// TwinCAT 3 PLC project AD_DA
// ProgramVersion: 3.1.4020.2
// libraries:
//   Tc2_Standard, * (Beckhoff Automation GmbH)
//   Tc2_System, * (Beckhoff Automation GmbH)
//   Tc3_Module, * (Beckhoff Automation GmbH)
// project tree:
//   FB_Lib/FB_ActionneurSimple/ FB_ActionneurSimple.TcPOU, ST_Erreur.TcDUT, ST_ParamActionneur.TcDUT
//   FB_Lib/ FB_analo_and_digital.TcPOU, FB_Etape.TcPOU
//   FB_Lib/FB_GestionModes/ FB_Btn.TcPOU, FB_CycleAuto.TcPOU, FB_CycleInit.TcPOU, FB_CycleMan.TcPOU, FB_MMA.TcPOU, p_InitVar.TcPOU
//   FB_Lib/FB_GestionModes/IO/ ST_IO.TcDUT, ST_IOInput.TcDUT, ST_IOInputSimul.TcDUT, ST_IOOutput.TcDUT, ST_IOOutputSimul.TcDUT
//   FB_Lib/FB_GestionModes/Param/ E_ModeMMA.TcDUT, ST_Param.TcDUT, ST_ParamFixed.TcDUT, ST_ParamRecipe.TcDUT, ST_ParamStatus.TcDUT
//   GVLs/ GVL.TcGVL
//   / PlcTask.TcTTO
//   POUs/ MAIN.TcPOU
// (motion and I/O tree: see PLC project 1calcul)
// real-time tasks:
//   TASK PlcTask: cycle T#1ms, priority 20, ADS port 350
// variable links:

CONFIGURATION AD_DA
    RESOURCE PLC ON TwinCAT3
        TASK PlcTask(INTERVAL := T#10ms, PRIORITY := 20);
        PROGRAM MAIN WITH PlcTask : MAIN;
    END_RESOURCE
END_CONFIGURATION

// ---- FB_Lib/FB_ActionneurSimple/ST_Erreur.TcDUT
TYPE ST_Erreur :
STRUCT
	xState:BOOL; 		//shows the current error state
	iId : INT; 			//error number currently active
	sMessage : STRING; 	//error message for the active error
END_STRUCT
END_TYPE

// ---- FB_Lib/FB_ActionneurSimple/ST_ParamActionneur.TcDUT
TYPE ST_ParamActionneur :
STRUCT
	tTimeOut : TIME; 			//max time allowed for moving to position bevor xState=TRUE
	xPresenceSensOut : BOOL; 	//If at the out-pos a Sensor is available
	xPresenceSensIn : BOOL; 	//If at the in-pos a Sensor is availaible
	tMoveOutTimeDelay : TIME; 	//delay after activating xPresenceSensOut before turning off output. When there is no Sensor, only this time will be used.
	tMoveInTimeDelay : TIME; 	//delay after activating xPresenceSensIn before turning off output. When there is no Sensor, only this time will be used.
END_STRUCT
END_TYPE

// ---- FB_Lib/FB_GestionModes/IO/ST_IO.TcDUT
TYPE ST_IO :
STRUCT
	stIn:ST_IOInput;
	stOut:ST_IOOutput;
END_STRUCT
END_TYPE

// ---- FB_Lib/FB_GestionModes/IO/ST_IOInput.TcDUT
TYPE ST_IOInput :
STRUCT
	IxAruIO AT%I*  :BOOL;
	xStartIO AT%I* :BOOL;
	xStopIO AT%I*  :BOOL;
	xResetIO AT%I* :BOOL;
	xAuto AT%I* : BOOL;
	xManual AT%I* : BOOL;
END_STRUCT
END_TYPE

// ---- FB_Lib/FB_GestionModes/IO/ST_IOInputSimul.TcDUT
TYPE ST_IOInputSimul :
STRUCT
	IxAru :BOOL;
END_STRUCT
END_TYPE

// ---- FB_Lib/FB_GestionModes/IO/ST_IOOutput.TcDUT
TYPE ST_IOOutput :
STRUCT
	QxLampeRouge AT%Q*:BOOL;
	QxLampeVerte AT%Q* : BOOL;
	QxLampeOrange AT%Q* :BOOL;
END_STRUCT
END_TYPE

// ---- FB_Lib/FB_GestionModes/IO/ST_IOOutputSimul.TcDUT
TYPE ST_IOOutputSimul :
STRUCT
	QxLampeRouge AT%Q*:BOOL;
END_STRUCT
END_TYPE

// ---- FB_Lib/FB_GestionModes/Param/E_ModeMMA.TcDUT

TYPE E_ModeMMA :
(
	Init := 0,
	Auto,
	Man
);
END_TYPE

// ---- FB_Lib/FB_GestionModes/Param/ST_Param.TcDUT
TYPE ST_Param :
STRUCT
	stStatus:ST_ParamStatus;//informations d'états (compteur de pièces, modes,...)
	stFixed:ST_ParamFixed;//Paramètres pas en lien avec le produit, fixe
	stRecipe:ST_ParamRecipe;//Paramètres en lien avec le produit
END_STRUCT
END_TYPE

// ---- FB_Lib/FB_GestionModes/Param/ST_ParamFixed.TcDUT
TYPE ST_ParamFixed :
STRUCT
END_STRUCT
END_TYPE

// ---- FB_Lib/FB_GestionModes/Param/ST_ParamRecipe.TcDUT
TYPE ST_ParamRecipe :
STRUCT
	
END_STRUCT
END_TYPE

// ---- FB_Lib/FB_GestionModes/Param/ST_ParamStatus.TcDUT
TYPE ST_ParamStatus :
STRUCT
	eMMA : E_ModeMMA; 
	xModePasAPas:BOOL;
	xErreur:BOOL;
	xInitOk:BOOL;//indique que l'initialisation a été exécutée
END_STRUCT
END_TYPE

// ---- GVLs/GVL.TcGVL
{attribute 'qualified_only'}
VAR_GLOBAL

END_VAR

// ---- POUs/MAIN.TcPOU
PROGRAM MAIN
VAR
	trans:FB_analo_and_digital;
	temp: LREAL;
	consigneMot : LREAL;
	motspeed : INT;
END_VAR
VAR_INPUT
	Read AT%I* : INT;
	ReadPot AT%I* : INT;
END_VAR
VAR_OUTPUT
	Write AT%Q* : INT;
	Motor AT%Q* : INT;
END_VAR

IF(consigneMot<trans.oRAWValue) THEN
	motspeed:=motspeed-20;
END_IF
IF(consigneMot>trans.oRAWValue) THEN
	motspeed:=motspeed+20;
END_IF

//Motor:=motspeed;

//read value fromPot and transform it into a value from -10 to 10Volt
trans(iRAWValue:=Read,iResolution:=16,iValMin:=-30,iValMax:=30,iValInputMin:=-10,iValInputMax:=10,iTransToPhysical:=TRUE);
temp:=trans.oPhysicalValue;
//take the temporary variable and stretch it to 3.4 max value. write it to the display
trans(iPhysicalValue:=temp,iResolution:=16,iValMin:=10,iValMax:=10,iTransToPhysical:=FALSE);
write:=LREAL_TO_INT(trans.oRAWValue);

END_PROGRAM

// ---- FB_Lib/FB_analo_and_digital.TcPOU
FUNCTION_BLOCK FB_analo_and_digital
VAR_INPUT
	iRAWValue : LREAL;				//raw Value read from sensor (registre)
	iResolution : INT; 				//resolution in bits
	iValMin: LREAL;					//min physical value possible
	iValMax: LREAL;					//max physical value possible
	iTransToPhysical : BOOL;		//RAW --> Physical when TRUE
	iValInputMax: LREAL;			//max input value at the Box--> normaly -10 to 10V
	iValInputMin: LREAL;			//min input value at the Box--> normaly -10 to 10V
	iPhysicalValue : LREAL;			//valeur physique
END_VAR
VAR_OUTPUT
	oPhysicalValue : LREAL;			//valeur physique sur l'entree de l'input
	oInputValue : LREAL;			//valeur physique sur l'entree de l'input dans la plage de ValInputMax / min
	oRAWValue : LREAL;				//raw Value read from sensor (registre)
END_VAR
VAR	
	temp : LREAL;
	temp2 : LREAL;	
END_VAR

temp2:=expt(2,iResolution);



IF(iTransToPhysical) THEN
	//RAW Input to physical value
	temp:=(iValInputMax-iValInputMin) / temp2;
	oInputValue:=iValInputMin + (temp * (iRAWValue + temp2/2));
	
	
	temp:=(iValMax-iValMin) / temp2;
	oPhysicalValue:=iValMin + (temp * (iRAWValue+temp2/2));
ELSE
	//Physical value to raw-Value
	temp:=(iValMax-iValMin) / temp2;
	oRAWValue:= iValMin+ (iPhysicalValue / temp);
			
END_IF

END_FUNCTION_BLOCK

// ---- FB_Lib/FB_ActionneurSimple/FB_ActionneurSimple.TcPOU
FUNCTION_BLOCK FB_ActionneurSimple
VAR_INPUT
	xInGoOut AT%I*:BOOL;				//input for going out
	xInGoIn AT%I*:BOOL;					//input for going in
	xReset AT%I*:BOOL;					//Reset all (go back to init state
	
	xAutorizeOut AT%I* : BOOL;		//allowed to do the move requested with xInGoOut, If this is false Programm will threw an error
	xAutorizeIn At%I* : BOOL;			//allowed to do the move requested with xInGoIn, If this is false Programm will threw an error
	
	stParam:ST_ParamActionneur;	//Param for actuator 
END_VAR
VAR_OUTPUT
	xInOutPos:BOOL;
	xInInPos:BOOL;
	
	xGoingOutNow AT%Q*:BOOL; //indication that actor is going in Out-Pos
	xGoingInNow AT%Q*:BOOL; //indication that actor is going in In-Pos
	
	QxOutOutput AT%Q*:BOOL;//Output to actuator for going Out
	QxInOutput AT%Q*:BOOL;//Output to actuator for going In
	
	IxSensOut AT%I*:BOOL;	//Sensor for the reached In-Pos
	IxSensIn AT%I*:BOOL;//Sensor for the reached Out-Pos
		
	stError:ST_Erreur;//Error Struct
	
	QxVanneDeBloquage AT%Q* : BOOL; //Vanne de blocace. Elle devient seulement 1 si l'autorisation entree/sortie est present
END_VAR
VAR
	fbEtape:FB_Etape;
	fbTimeOut:TON;
	fbRTrigOut:R_Trig;
	fbRTrigIn:R_Trig;
		
	

END_VAR

fbEtape.mActualisation(xModeStepForStep,xNextStep);

//check rising edges on 
fbRTrigOut(clk:=xInGoOut);
fbRTrigIn(clk:=xInGoIn);

//Go to the next step when there is an Out-Command
IF fbRTrigOut.Q AND NOT(fbEtape.iNo>=200 AND fbEtape.iNo<=299) THEN	//When rising-edge was detected
	IF xAutorizeOut THEN
		fbEtape.piVal:=200;
	ELSE
		stError.iId:=10;
		stError.sMessage:='Autorisation refusee pour action sortir verin';
	END_IF		
fbEtape.piVal:=200;	
END_IF

//Go to the next step when there is an In-Command
IF fbRTrigIn.Q AND NOT(fbEtape.iNo>=100 AND fbEtape.iNo<=199) THEN	//When rising-edge was detected and not already going In
	IF xAutorizeIn THEN
		fbEtape.piVal:=100;
	ELSE
		stError.iId:=11;
		stError.sMessage:='Autorisation refusee pour action rentrer verin';
	END_IF	
END_IF

//Reset
IF xReset THEN
	fbEtape.piVal:=0;
	stError.xState:=0;
	xInOutPos:=0;
	xInInPos:=0;
END_IF

//check pour vanne de blocage
QxVanneDeBloquage:= (xAutorizeOut OR xAutorizeIn);

//Reset de l'erreur
IF stError.xState THEN
	stError.iId:=0;
	stError.sMessage:='';
END_IF



CASE fbEtape.iNo OF
	0:fbEtape.psMess:='Wait for an In or Out command';
	//-----------------------------------------------
	100:fbEtape.psMess:='Action go In';
		IF xAutorizeIn THEN
			fbEtape.piVal:=110;
			fbEtape.tTimeQ:=stParam.tMoveInTimeDelay;
		END_IF
	110:fbEtape.psMess:='Going in, waiting for IxSensIn';
		IF (IxSensIn AND stParam.xPresenceSensIn) OR NOT stParam.xPresenceSensIn THEN
			fbEtape.piVal:=150;
		END_IF
	150:fbEtape.psMess:='Action rentre, attend tenps d enveloppe';
		IF fbEtape.xTimeQ THEN
			fbEtape.piSVal:=199;
		END_IF
	199:fbEtape.psMess:='In-Position reached';
		IF (NOT IxSensIn) AND stParam.xPresenceSensIn THEN
			fbEtape.piVal:=150;
		END_IF
	//-----------------------------------------------
	200:fbEtape.psMess:='Action go Out';
		IF xAutorizeOut THEN
			fbEtape.piVal:=210;
			fbEtape.tTimeQ:=stParam.tMoveInTimeDelay;
		END_IF
	210:fbEtape.psMess:='Going Out, waiting for IxSensOut';
		IF (IxSensOut AND stParam.xPresenceSensOut) OR NOT stParam.xPresenceSensOut THEN
			fbEtape.piVal:=250;
		END_IF
	250:fbEtape.psMess:='Action sort, attend temps d enveloppe';
		IF fbEtape.xTimeQ THEN
			fbEtape.piSVal:=299;
		END_IF
	299:fbEtape.psMess:='Out-Pos reached';
		IF (NOT IxSensOut) AND stParam.xPresenceSensoUT THEN
			fbEtape.piVal:=250;
		END_IF
	
	999:fbEtape.psMess:='Erreur';
END_CASE

//Activation du Timer
fbTimeOut(IN:=(fbEtape.iNo>100 AND fbEtape.iNo<199 OR fbEtape.iNo>200 AND fbEtape.iNo<299)
				AND (NOT fbRTrigIn.Q AND NOT fbRTrigOut.Q),PT:=stParam.tTimeOut);	


(*Liste des erreurs possibles :
-	10 Si un ordre de déplacement sort est donné et que l’entrée, xAutoriseSort n’est pas vrai, on indique une erreur
-	11 Idem pour xAutoriseRentre
-	20 Erreur de timeout sort
-	21 Erreur de timeout rentre
-	30 Les deux fins de course sont vraies en même temps
-	31 Double consignes, xSetSort=1 et xSetRentre=1*)				
//Gestion des erreurs
IF fbTimeOut.Q THEN
	IF fbEtape.iNo < 200 THEN
		stError.sMessage:='Erreur de timeout rentre';
		stError.iId:=21;
	ELSIF fbEtape.iNo>200 THEN
		stError.sMessage:='Erreur de timeout sort';
		stError.iId:=20;
	END_IF
ELSIF IxSensIn AND IxSensOut THEN
	stError.sMessage:='Les deus fins de course sont vraies en même temps';
	stError.iId:=30;
ELSIF xInGoOut AND xInGoIn THEN
	stError.sMessage:='Double consigne,xSetSort=1 et xSetRentre=1';
	stError.iId:=31;
END_IF

stError.xState :=fbEtape.iNo=999 OR fbTimeOut.Q OR (IxSensIn AND IxSensOut) OR (xInGoIn AND xInGoOut);


//Activation des états
xInInPos:=fbEtape.iNo=199;
xInOutPos:=fbEtape.iNo=299;
xGoingInNow:= QxInOutput AND NOT IxSensIn;
xGoingOutNow:= QxOutOutput AND NOT IxSensOut;


//Activation des sorties
QxOutOutput:=fbEtape.iNo>200 AND fbEtape.iNo<=299;
QxInOutput:=fbEtape.iNo>100 AND fbEtape.iNo<=199;

END_FUNCTION_BLOCK

// ---- FB_Lib/FB_Etape.TcPOU
FUNCTION_BLOCK FB_Etape
VAR_INPUT
	tTimeQ :TIME;			//Time to stay in one state after which xTimeQ will go to TRUE
END_VAR
VAR_OUTPUT
	tTimeState: TIME ; 	//passed time in the actual state
	xTimeQ : BOOL ;		//is TRUE when time passed in the actual State is greather then tTimeQ
	xTransition:BOOL; 	//information that the state has just changed. For use when entering a new State the first time
	iNo:INT:=0; 		//State number running at the moment
	sMess :STRING ; 	//Information message about the current running state
END_VAR
VAR
	iMemNo:INT;				//Used for xTransition. Saves the actual state of the machine
	fbTon:ton;				//Timer for the actual State
	fbRtrig:R_trig;			//detector for rising edges
	xMemModeStepByStep:BOOL;	//Mem for the actual running Mode (see method mActualisation)
	
END_VAR

//executed at each state-machine-loop
METHOD PUBLIC mActualisation
VAR_INPUT
	xModeStepByStep: BOOL; //activate the Stepping-Mode (TRUE=ON)
	xSetNextStep: BOOL; //go to the next Step on rising eddge
END_VAR
//manage StepByStep
//-----------------

//Detect rising edge
fbRtrig(CLK:=xSetNextStep);
//copy the mode input to use it in piSVal
xMemModeStepByStep:=xModeStepByStep;

//detect a state changement in the state machine
xTransition:=iNo<>iMemNo;

//start Method when the state has changed
IF xTransition THEN
	mTransition();
END_IF

//manage the Timer and associated Variabels
//-----------------------------------------
fbTON(IN:=(iNo=iMemNo), PT:=T#71582M47S295MS, ET=>tTimeState); //will be resetted when the state is changed

//going to TRUE when longer in the actual State than tTimeQ
xTimeQ:=(tTimeState>=tTimeQ);

//save the last running state
iMemNo:=iNo;
END_METHOD

//Executed when a State has changed
METHOD PRIVATE mTransition
//make a new String to display
sMess:=CONCAT('iNo:=',int_to_string(iNo));
END_METHOD

//going to the next step while paying attention to StepByStep Mode
PROPERTY PUBLIC piSVal : INT
SET
IF NOT xMemModeStepByStep THEN
	//Step by step mode is off
	iNo:=piSVal;
	ELSIF fbRtrig.Q THEN
		//a button press on "xSetNextStep" has been detected
		iNo:=piSVal;
END_IF
END_SET
END_PROPERTY

//going to the next step without paying attention to StepByStep Mode
PROPERTY PUBLIC piVal : INT
SET
//set the next step
iNo:=piVal;
END_SET
END_PROPERTY

//
PROPERTY PUBLIC psMess : STRING
SET
//write the description of the actual step to sMess
IF xTransition THEN
	sMess:=psMess;
END_IF
END_SET
END_PROPERTY

END_FUNCTION_BLOCK

// ---- FB_Lib/FB_GestionModes/FB_Btn.TcPOU
FUNCTION_BLOCK FB_Btn
VAR_INPUT
	xStart:BOOL;
	xStop:BOOL;
	xReset:BOOL;
	xNextPas:BOOL;
	xAru:BOOL;
	
	xManAct1Rentre: BOOL;
	xManAct1Sort : BOOL;
	
	xManAct2Rentre: BOOL;
	xManAct2Sort : BOOL;
	
	xManAct3Rentre: BOOL;
	xManAct3Sort : BOOL;
END_VAR
VAR_OUTPUT
END_VAR
VAR
END_VAR

END_FUNCTION_BLOCK

// ---- FB_Lib/FB_GestionModes/FB_CycleAuto.TcPOU
FUNCTION_BLOCK FB_CycleAuto
VAR_INPUT
	xStart:BOOL;
	xStop:BOOL;
	xReset:BOOL;
END_VAR
VAR_OUTPUT
	fbRtrigStart:R_trig;
	xBusy:BOOL;
	xMemStop:BOOL:=FALSE;
	iEtape:INT;
END_VAR
VAR
	fbEtape:FB_Etape;
END_VAR

fbEtape.mActualisation(stParam.stStatus.xModePasAPas,fbBtn.xNextPas);

fbRtrigStart(clk:=xStart);

IF xStop THEN
	xMemStop:=TRUE;
END_IF

IF xReset THEN
	fbEtape.piVal:=0;
END_IF

CASE fbEtape.iNo OF
	0:IF fbRtrigStart.Q THEN
		xMemStop:=FALSE;
		fbEtape.piVal:=100;
	END_IF
	100:fbEtape.psMess:='fonction allume lampe1';
		//assigne le temps de comptage
		fbEtape.tTimeQ:=T#2S;
		fbEtape.piVal:=110;
	110:fbEtape.psMess:='activation compteur 2s - attendre fin comptage';
		IF fbEtape.xTimeQ THEN
			fbEtape.piSVal:=120;
		END_IF
	120:fbEtape.psMess:='Actionneur1 sort';
		IF fbAct1.xInOutPos THEN
			fbEtape.piSVal:=121;
		END_IF
	121:fbEtape.psMess:='Actionneur2 sort';
		IF fbAct2.xInOutPos THEN
			fbEtape.piSVal:=122;
		END_IF
	122:fbEtape.psMess:='Actionneur3 sort';
		IF fbAct3.xInOutPos THEN
			fbEtape.piSVal:=130;
		END_IF
	130:fbEtape.psMess:='Actionneur3 rentre';
		IF fbAct3.xInInPos THEN
			fbEtape.piSVal:=131;
		END_IF
	131:fbEtape.psMess:='Actionneur2 rentre';
		IF fbAct2.xInInPos THEN
			fbEtape.piSVal:=132;
		END_IF
	132:fbEtape.psMess:='Actionneur1 rentre';
		IF fbAct1.xInInPos THEN
			fbEtape.piSVal:=200;
		END_IF
	200:fbEtape.psMess:='fonction allume lampe1';
		//assigne le temps de comptage
		fbEtape.tTimeQ:=T#1S;
		fbEtape.piVal:=210;
	210:fbEtape.psMess:='activation compteur 1s - attendre fin comptage';
		IF fbEtape.xTimeQ THEN
			fbEtape.piSVal:=300;
		END_IF
	300:fbEtape.psMess:='fonction lampes off';
		//assigne le temps de comptage
		fbEtape.tTimeQ:=T#2S;
		fbEtape.piVal:=310;
	310:fbEtape.psMess:='activation compteur 2s - attendre fin comptage';
		IF fbEtape.xTimeQ THEN
			fbEtape.piSVal:=900;
		END_IF
	900:fbEtape.psMess:='Test si demande arrrêt en fin de cycle';
		IF xMemStop THEN
		fbEtape.piSVal:=999;
		ELSE
		fbEtape.piSVal:=100;
	END_IF
	999:fbEtape.psMess:='FIN';
		fbEtape.piSVal:=0;
END_CASE

xBusy:=fbEtape.iNo<>0;
iEtape:=fbEtape.iNo;

END_FUNCTION_BLOCK

// ---- FB_Lib/FB_GestionModes/FB_CycleInit.TcPOU
FUNCTION_BLOCK FB_CycleInit
VAR_INPUT
	xStart : BOOL;
	xStop : BOOL;
END_VAR
VAR_OUTPUT
	fbRtrigStart:R_trig;
	xBusy:BOOL;
	iEtape:INT;
END_VAR
VAR
	fbEtape:FB_Etape;
END_VAR

fbEtape.mActualisation(stParam.stStatus.xModePasAPas,fbBtn.xNextPas);

fbRtrigStart(clk:=fbBtn.xStart);


CASE fbEtape.iNo OF
	0:fbEtape.psMess:='Attendre - Pret';
		IF xStart THEN
			fbEtape.piVal:=99;
		END_IF
	99: fbEtape.psMess:='Reset sur les Actionneurs';
		fbEtape.piSVal:=100;
		
	100:fbEtape.psMess:='Initialiser les positions';
		IF  fbAct1.xInInPos AND fbAct2.xInInPos AND NOT fbAct3.xInInPos THEN
			fbEtape.piSVal:=999;
		END_IF
	
	999:fbEtape.psMess:='Fin Cycle Init - Attente de Stop';
		IF (xStop) THEN
		fbEtape.piSVal:=0;
	END_IF
END_CASE

xBusy:=fbEtape.iNo<>0;
iEtape:=fbEtape.iNo;

END_FUNCTION_BLOCK

// ---- FB_Lib/FB_GestionModes/FB_CycleMan.TcPOU
FUNCTION_BLOCK FB_CycleMan
VAR_INPUT
	xStart : BOOL;
	xStop : BOOL;
	
	
END_VAR
VAR_OUTPUT
	fbRtrigStart:R_trig;
	xBusy:BOOL;
	iEtape:INT;
END_VAR
VAR
	fbEtape:FB_Etape;
END_VAR

fbEtape.mActualisation(stParam.stStatus.xModePasAPas,fbBtn.xNextPas);

fbRtrigStart(clk:=fbBtn.xStart);


CASE fbEtape.iNo OF
	0:	fbEtape.psMess:='Attendre - Pret';
		IF xStart THEN
			fbEtape.piVal:=100;
		END_IF
	100:fbEtape.psMess:='Selectioner quoi faire';
		//changer de mode
		IF  stParam.stStatus.eMMA<>Man THEN
			fbEtape.piSVal:=990;
		END_IF
		//Act1:
		IF (fbBtn.xManAct1Rentre) THEN
			fbEtape.piVal:=201;
		END_IF
		IF (fbBtn.xManAct1Sort) THEN
			fbEtape.piVal:=202;
		END_IF
		//Act2:
		IF (fbBtn.xManAct2Rentre) THEN
			fbEtape.piVal:=203;
		END_IF
		IF (fbBtn.xManAct2Sort) THEN
			fbEtape.piVal:=204;
		END_IF
		//Act3:
		IF (fbBtn.xManAct3Rentre) THEN
			fbEtape.piVal:=205;
		END_IF
		IF (fbBtn.xManAct3Sort) THEN
			fbEtape.piVal:=206;
		END_IF
		
		
		
	201: fbEtape.psMess:='Action : Act 1 Rentre';
		IF (NOT fbBtn.xManAct1Rentre) THEN
			fbEtape.piVal:=100;
		END_IF
	202: fbEtape.psMess:='Action : Act 1 Sort';
		IF (NOT fbBtn.xManAct1Sort) THEN
			fbEtape.piVal:=100;
		END_IF
	203: fbEtape.psMess:='Action : Act 2 Rentre';
		IF (NOT fbBtn.xManAct2Rentre) THEN
			fbEtape.piVal:=100;
		END_IF
	204: fbEtape.psMess:='Action : Act 2 Sort';
		IF (NOT fbBtn.xManAct2Sort) THEN
			fbEtape.piVal:=100;
		END_IF
	205: fbEtape.psMess:='Action : Act 3 Rentre';
		IF (NOT fbBtn.xManAct3Rentre) THEN
			fbEtape.piVal:=100;
		END_IF
	206: fbEtape.psMess:='Action : Act 3 Sort';
		IF (NOT fbBtn.xManAct3Sort) THEN
			fbEtape.piVal:=100;
		END_IF
	
	990:fbEtape.psMess:='Finir Cycle Man';
		//ici on fait des choses de fin (ex. eteindre un moteur qui tourne encore)
		IF (1) THEN
			fbEtape.piSVal:=999;
		END_IF	
	999:fbEtape.psMess:='Fin Cycle Manuel';
		IF (xStop) THEN
			fbEtape.piSVal:=0;
		END_IF
		
END_CASE

xBusy:=fbEtape.iNo<>0;
iEtape:=fbEtape.iNo;

END_FUNCTION_BLOCK

// ---- FB_Lib/FB_GestionModes/FB_MMA.TcPOU
FUNCTION_BLOCK FB_MMA
VAR_INPUT
END_VAR
VAR_OUTPUT
	iEtape:INT;
END_VAR
VAR
	fbEtape:FB_Etape;
	p_InitVar : p_InitVar;
END_VAR

fbEtape.mActualisation(FALSE,FALSE);

//on active l'arret d'urgence si l'entree devient false
IF NOT fbBtn.xAru AND fbEtape.iNo>10 AND fbEtape.iNo<800 THEN
	fbEtape.piVal:=900; 
END_IF

//on fait un reset
IF fbBtn.xReset AND fbEtape.iNo>10 AND fbEtape.iNo<800 THEN
	fbEtape.piVal:=800;
END_IF


CASE fbEtape.iNo OF
	0://mise en marche du système
		fbEtape.piVal:=10;
	
	10://OB100 Siemens
		p_InitVar(); //initialiser les vars (propre a la machine)
		fbEtape.piVal:=50;
	
	50:fbEtape.psMess:='Selection du mode MMA';
		IF (stParam.stStatus.eMMA=Auto) THEN
			fbEtape.piVal:=300;
		ELSIF (stParam.stStatus.eMMA=Man) THEN
			fbEtape.piVal:=210;
		ELSIF (stParam.stStatus.eMMA=Init) THEN
			fbEtape.piVal:=100;
		END_IF
		
	//--------------------------------------------------------------
	//Init
	//--------------------------------------------------------------
	100:fbEtape.psMess:='Cycle Init | Attente de fbBtn.xStart';
		IF (fbBtn.xStart) THEN
			fbEtape.piVal:=110;
		ELSIF (stParam.stStatus.eMMA<>Init) THEN
			fbEtape.piVal:=50;
		END_IF
	110:fbEtape.psMess:='Cycle Init | Attente fin';
		IF fbCycleInit.iEtape=999 THEN
		fbEtape.piVal:=50;
		END_IF
	111:fbEtape.psMess:='Cycle Init | Finir';
		IF fbCycleInit.xBusy THEN
		fbEtape.piVal:=50;
		END_IF
		
	//--------------------------------------------------------------
	//Manual
	//--------------------------------------------------------------
	210:fbEtape.psMess:='Cycle Manuel | Attente de changement de mode';
		IF (fbCycleMan.iEtape=999) THEN
		fbEtape.piVal:=211;
		END_IF
	211:fbEtape.psMess:='Cycle Manuel | Finir';
		IF (fbCycleMan.xBusy) THEN
		fbEtape.piVal:=50;
		END_IF
		
	//--------------------------------------------------------------
	//Auto
	//--------------------------------------------------------------
	300:fbEtape.psMess:='Mode Auto | Attente de fbBtn.xStart';
		IF (fbBtn.xStart) THEN
			fbEtape.piVal:=340;
		ELSIF (stParam.stStatus.eMMA<>Auto) THEN
			fbEtape.piVal:=50;
		END_IF
	
	340:fbEtape.psMess:='Mode Auto | Cycle Init - attente fin';
		//si le cycle INIT est terminé alors on continue
		fbEtape.piVal:=341;
		
	341:fbEtape.psMess:='Mode Auto | Cycle Init - Finir';
		//si le cycle INIT est terminé alors on continue
		IF fbCycleInit.iEtape=999 THEN
			fbEtape.piVal:=350;
		END_IF
		
	350:fbEtape.psMess:='Mode Auto | Production - attend signal Stop';
		IF (fbBtn.xStop OR stParam.stStatus.xErreur ) THEN 
			fbEtape.piVal:=390;
		END_IF
		
	390:fbEtape.psMess:='Mode Auto | Attendre fin';
		IF (NOT fbCycleAuto.xBusy) THEN
			fbEtape.piVal:=50;
		END_IF
		
	//--------------------------------------------------------------
	//Reset
	//--------------------------------------------------------------
	800:fbEtape.psMess:='Reset | Procédure de reset, stop imédiat';
		fbEtape.piVal:=810;
	810:fbEtape.psMess:='Reset | Ordre pour pilotage reste sur cycle';
		fbEtape.piVal:=899;
	899:fbEtape.psMess:='Reset | Fin de procédure Reset';
		fbEtape.piVal:=50;
		
	//--------------------------------------------------------------
	//ARU
	//--------------------------------------------------------------
	900:fbEtape.psMess:='ARU | Procédure de ARU';
		fbEtape.piVal:=910;
	910:fbEtape.psMess:='ARU | Ordre pour pilotage reste sur cycle';
		fbEtape.piVal:=950;
	950:fbEtape.psMess:='ARU | ok - Attente de quittance';
		IF fbBtn.xAru THEN
			fbEtape.piVal:=999;
	END_IF
	999:fbEtape.psMess:='ARU | Fin de procédure ARU';
		fbEtape.piVal:=50;
END_CASE


iEtape:=fbEtape.iNo;

END_FUNCTION_BLOCK

// ---- FB_Lib/FB_GestionModes/p_InitVar.TcPOU
FUNCTION_BLOCK p_InitVar
VAR_INPUT
END_VAR
VAR_OUTPUT
END_VAR
VAR
	tEnvStabSort: INT;
END_VAR

fbAct1.stParam.xPresenceSensIn:=TRUE;
fbAct1.stParam.xPresenceSensOut:=TRUE;
fbAct1.stParam.tTimeOut:=T#10S;
fbAct1.stParam.tMoveInTimeDelay:=T#1.5S;
fbAct1.stParam.tMoveOutTimeDelay:=T#1.5S;

fbAct2.stParam.xPresenceSensIn:=TRUE;
fbAct2.stParam.xPresenceSensOut:=TRUE;
fbAct2.stParam.tTimeOut:=T#10S;
fbAct2.stParam.tMoveInTimeDelay:=T#1.5S;
fbAct2.stParam.tMoveOutTimeDelay:=T#1.5S;

fbAct3.stParam.xPresenceSensIn:=FALSE;
fbAct3.stParam.xPresenceSensOut:=TRUE;
fbAct3.stParam.tTimeOut:=T#10S;
fbAct3.stParam.tMoveInTimeDelay:=T#3S;
fbAct3.stParam.tMoveOutTimeDelay:=T#1.5S;

stParam.stStatus.eMMA:=Init;

END_FUNCTION_BLOCK
